RoboDK station: 2. doosan_waypoint_patrol.rdk

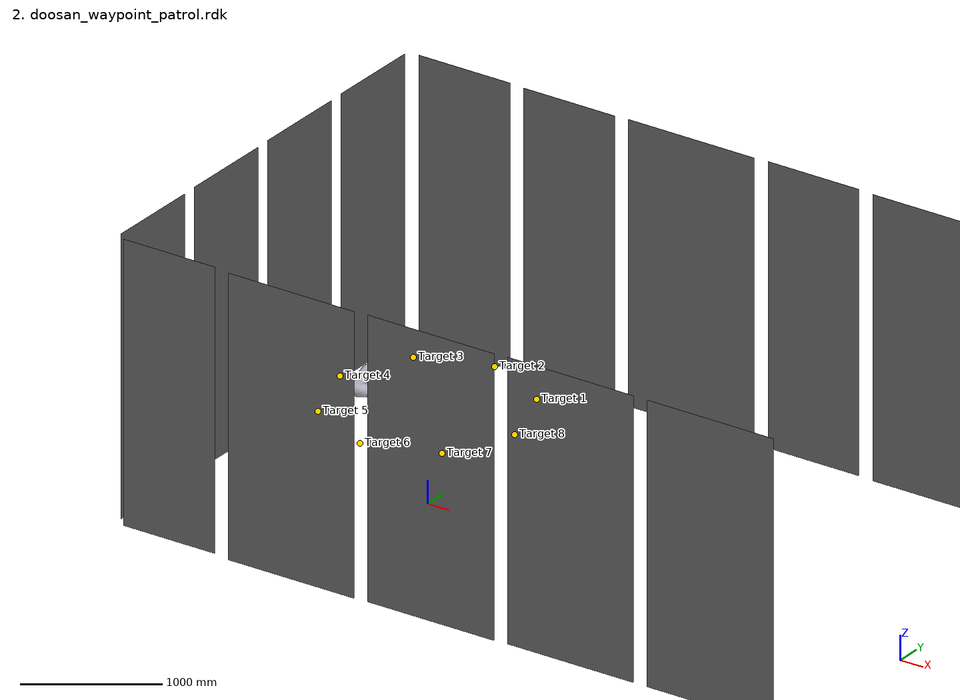
[picture v0: the station drawn from its stored meshes, robots at their saved joint values, targets as dots, program paths as lines]
Station 2. doosan_waypoint_patrol (saved by RoboDK 5.9.6). Poses are relative to the parent item; angles as X-Y-Z fixed-axis rotations.
  - frame Doosan M1013 Base at (0, 0, 0) mm
    - robot Doosan M1013: 6 axes, payload 10 kg, reach 1300 mm, repeatability 0.1 mm, weight 33 kg
        modified DH rows (alpha deg, a mm, theta deg, d mm): 0, 0, 0, 152.5; -90, 0, -90, -34.506; 0, 620, -90, 0; -90, 0, 0, 559; 90, 0, 0, 0; -90, 0, 180, 121
        joint limits [-360, -360, -160, -360, -360, -360] to [360, 360, 160, 360, 360, 360]; home [0, 0, 90, 0, 0, 0]; saved at [190.519, 0, 90, -17.888, 0, 17.888]
      - tool Zivid On-Arm Extender OA02E, TCP at (0, 0.06, 95.34) mm, size 92 x 91.8 x 80 mm
        - object Intel RealSense D435 Camera at (0, 0, 0) mm, size 89.8 x 25 x 25.1 mm, geometry from Intel-RealSense-D435-Camera.sld
    - target Target 1 (Cartesian target) at (572.61, 523.89, 772.5) mm, rotated rx 0 ry 90 rz 45 deg; joints [45, 0, 90, 0, 0, 0] of Doosan M1013
    - target Target 2 (Cartesian target) at (34.45, 775.34, 772.5) mm, rotated rx 0 ry 90 rz 90 deg; joints [90, 0, 90, 0, 0, 0] of Doosan M1013
    - target Target 3 (Cartesian target) at (-523.89, 572.61, 772.5) mm, rotated rx 0 ry 90 rz 135 deg; joints [135, 0, 90, 0, 0, 0] of Doosan M1013
    - target Target 4 (Cartesian target) at (-775.34, 34.45, 772.5) mm, rotated rx 0 ry 90 rz 180 deg; joints [180, 0, 90, 0, 0, 0] of Doosan M1013
    - target Target 5 (Cartesian target) at (-572.61, -523.89, 772.5) mm, rotated rx 0 ry 90 rz -135 deg; joints [301.091, -82.684, 68.126, -76.521, 93.464, -14.149] of Doosan M1013
    - target Target 6 (Cartesian target) at (-34.45, -775.34, 772.5) mm, rotated rx 0 ry 90 rz -90 deg; joints [270, -81.809, 99.801, 0, 72.007, 0] of Doosan M1013
    - target Target 7 (Cartesian target) at (523.89, -572.61, 772.5) mm, rotated rx 0 ry 90 rz -45 deg; joints [234.547, -83.929, 76.599, 80.53, 91.213, 7.23] of Doosan M1013
    - target Target 8 (Cartesian target) at (775.34, -34.45, 772.5) mm, rotated rx 0 ry 90 rz 0 deg; joints [360, 0, 90, 0, 0, 0] of Doosan M1013
  - camera Camera 1
  - Python program doosan_waypoint_patrol (listed below)
  - object Cell Safety Panels at (0, 0, 0) mm, size 5655.1 x 3636 x 2268 mm, geometry from Cell-Safety-Panels.sld
  - camera Camera 2

--- Python program doosan_waypoint_patrol ---
from robodk.robolink import Robolink, ITEM_TYPE_ROBOT, ITEM_TYPE_TARGET, RUNMODE_SIMULATE, StoppedError
import time

# -----------------------------
# Config
# -----------------------------
ROBOT_NAME = "Doosan M1013"
TARGET_PREFIX = "Target "
PAUSE_SECONDS = 1.5

# Keep running forever
LOOP_FOREVER = True

# Simulation/debug only (set False if you want collision checking ON)
DISABLE_COLLISION_CHECK = True

# -----------------------------
# Connect
# -----------------------------
RDK = Robolink()
RDK.setRunMode(RUNMODE_SIMULATE)

robot = RDK.Item(ROBOT_NAME, ITEM_TYPE_ROBOT)
if not robot.Valid():
    raise Exception(f"Robot '{ROBOT_NAME}' not found")

robot.setSpeedJoints(10)
robot.setAccelerationJoints(20)

# Try to disable collision checking (API differs by RoboDK version)
if DISABLE_COLLISION_CHECK:
    try:
        RDK.setCollisionActive(0)  # 0 = OFF, 1 = ON
        print("Collision checking disabled.")
    except Exception:
        try:
            RDK.Command("CollisionDetection", "Off")
            print("Collision checking disabled.")
        except Exception:
            print("Warning: Could not disable collision checking via API.")

# -----------------------------
# Build target list automatically: Target 1, Target 2, ...
# -----------------------------
targets = []
i = 1
while True:
    t = RDK.Item(f"{TARGET_PREFIX}{i}", ITEM_TYPE_TARGET)
    if not t.Valid():
        break
    targets.append(t)
    i += 1

if not targets:
    raise Exception("No targets found (expected names like 'Target 1', 'Target 2', ...)")

print(f"Robot '{ROBOT_NAME}' found. Moving through {len(targets)} targets in a loop...")

# -----------------------------
# Motion sequence
# -----------------------------
def run_sequence():
    for idx, target in enumerate(targets, start=1):
        print(f"Moving to {TARGET_PREFIX}{idx}")
        try:
            robot.MoveJ(target)  # or robot.MoveL(target)
            time.sleep(PAUSE_SECONDS)
        except StoppedError as e:
            print(f"Skipped {TARGET_PREFIX}{idx}: {e}")
        except Exception as e:
            print(f"Error on {TARGET_PREFIX}{idx}: {e}")

# Infinite loop
while LOOP_FOREVER:
    run_sequence()
